// TIA Portal V17 export
// export: Created 2023-03-22T09:29:52.1196935Z, ExportSetting WithDefaults, DisplayName Totally Integrated Automation Portal, DisplayVersion V17 Update 4, DisplayName TIA Portal Openness, DisplayVersion V17 Update 4, DisplayName TIA Portal Version Control Interface, DisplayVersion V17, DisplayName STEP 7 Professional, DisplayVersion V17 Update 4, DisplayName STEP 7 Safety, DisplayVersion V17, DisplayName WinCC Professional, DisplayVersion V17 Update 4
VAR_GLOBAL   // PLC tag table "Rack Variables"
   "Emergency stop from PCS1 (PE)" AT %I56.0 : Bool;   // xFDI_Slot02_In01_EPCS1
   "Emergency stop from PCS2 (PE) (future expansion)" AT %I56.4 : Bool;   // xFDI_Slot02_In02_EPCS2
   "Emergency stop from External (future expansion)" AT %I56.1 : Bool;   // xFDI_Slot02_In03_EExt
   "PWCLH0 Common mode signal" AT %I56.5 : Bool;   // xFDI_Slot02_In04_125A3
   "PWCRH0 Common mode signal" AT %I56.2 : Bool;   // xFDI_Slot02_In05_225A3
   "Spare(1)" AT %I56.6 : Bool;   // xFDI_Slot02_In06_Xxxxxx
   "Spare(2)" AT %I56.3 : Bool;   // xFDI_Slot02_In07_Xxxxxx
   "Spare(3)" AT %I56.7 : Bool;   // xFDI_Slot02_In08_Xxxxxx
END_VAR
